TYPE ST_CURING_STATION_HEATER_CONTROL_SERVICE :
STRUCT
	
END_STRUCT
END_TYPE

(* stored: Version 1.1.0.1
   DUT ST_CURING_STATION_HEATER_CONTROL_SERVICE: Id {36b3e498-0d47-4931-9c08-eda65c62a206} *)
